FUNCTION_BLOCK SEMA_VIEW
  (* Standard: 61499-1; Classification: HMI; Function: Output; Type: 4xLED *)
  (* Version 0.4, 2018-07-27, JHC, Holobloc Inc, Updated I/O documentation. *)
  (* Version 0.3, 2011-03-28, JHC, Holobloc Inc, Updated documentation. *)
  (* Version 0.2, 2008-11-10, JHC, Holobloc Inc, Moved to fb.rt.doc. *)
  (* Version 0.1, 2008-06-04, JHC, Holobloc Inc, Updated DOCTYPE. *)
  (* Version 0.0, 2001-02-21, JHC, Rockwell Automation *)
  PACKAGE fb.rt.DIAS;
  IMPORT fb.datatype.*;
  IMPORT fb.rt.*;
  IMPORT fb.rt.hmi.*;
  (* Compiler Java Sun JDK 1.7.0 *)
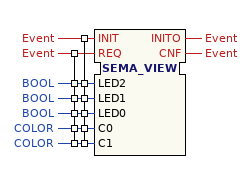
  EVENT_INPUT
    INIT WITH LED2, LED1, LED0, C0, C1; (* Initialize *)
    REQ WITH LED2, LED1, LED0, C0, C1; (* LED State/Color Update *)
  END_EVENT
  EVENT_OUTPUT
    INITO; (* INIT Confirm *)
    CNF; (* REQ Confirmation *)
  END_EVENT
  VAR_INPUT
    LED2 : BOOL;
    LED1 : BOOL;
    LED0 : BOOL; (* LSB - Least Significant Bit *)
    C0 : COLOR := COLOR#white; (* OFF color *)
    C1 : COLOR := COLOR#orange; (* ON color *)
  END_VAR
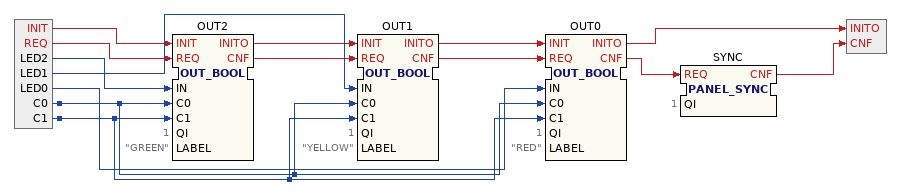
  FBS
    OUT2 : OUT_BOOL(QI := 1, LABEL := "GREEN");
    OUT1 : OUT_BOOL(QI := 1, LABEL := "YELLOW");
    OUT0 : OUT_BOOL(QI := 1, LABEL := "RED");
    SYNC : PANEL_SYNC(QI := 1); (* Synchronize frame buffer *)
  END_FBS
  EVENT_CONNECTIONS
    OUT2.INITO TO OUT1.INIT;
    OUT1.INITO TO OUT0.INIT;
    OUT0.INITO TO INITO;
    OUT2.CNF TO OUT1.REQ;
    OUT1.CNF TO OUT0.REQ;
    OUT0.CNF TO SYNC.REQ;
    SYNC.CNF TO CNF;
    INIT TO OUT2.INIT;
    REQ TO OUT2.REQ;
  END_CONNECTIONS
  DATA_CONNECTIONS
    LED2 TO OUT2.IN;
    LED1 TO OUT1.IN;
    LED0 TO OUT0.IN;
    C0 TO OUT2.C0;
    C0 TO OUT1.C0;
    C0 TO OUT0.C0;
    C1 TO OUT2.C1;
    C1 TO OUT1.C1;
    C1 TO OUT0.C1;
  END_CONNECTIONS
END_FUNCTION_BLOCK
